// TIA Portal V16 export
// export: Created 2024-12-03T15:41:41.4210961Z, ExportSetting WithDefaults, DisplayName Totally Integrated Automation Portal, DisplayVersion V16 Update 6, DisplayName TIA Portal Version Control Interface, DisplayVersion V16 Update 2, DisplayName TIA Portal Openness, DisplayVersion V16 Update 6, DisplayName TIA Portal Teamcenter Gateway, DisplayVersion V16, DisplayName SINAMICS Startdrive Advanced, DisplayVersion V16 Update 5, DisplayName SINAMICS Startdrive G130, G150, S120, S150, SINAMICS MV, S210, DisplayVersion V16 Update 5, DisplayName SINAMICS Startdrive G110M, G120, G120C, G120D, G120P, G115D, DisplayVersion V16 Update 5, DisplayName STEP 7 Professional, DisplayVersion V16 Update 6, DisplayName STEP 7 Safety, DisplayVersion V16, DisplayName WinCC Advanced / Unified PC, DisplayVersion V16 Update 6
FUNCTION_BLOCK "CM_Encoder_FB"   // FB119, SCL
{ S7_Optimized_Access := 'TRUE' }
VERSION : 0.1
// stored: AutoNumber true, IsIECCheckEnabled false, IsRetainMemResEnabled false, MemoryReserve 100, SetENOAutomatically false, UDAEnableTagReadback false
   VAR_INPUT
      dEncr : DInt;   // Encoder input
      dPPR : DInt;   // Number of pulses per revolution
      rDiameterWheel : Real;   // Diameter of the wheel driving the roller or belt conveyor (mm)
      rGearRatio : Real;   // GearRatio should be 1.0 for the standalone encoders
      x32or16bitEncr : Bool;   // 1 = 32 bit, 0 = 16 bit
   END_VAR
   VAR_IN_OUT
      IO_Encoder : "VirtualEncoder_UDT";
   END_VAR
   VAR
      d16bitEncr_Range : DInt := 65535;   // Range of 16 bit encoder (pulses)
      d32bitEncr_Range : DInt;   // Range of 32 bit encoder (pulses)
      dCheckRotationClockwise : DInt;
      rPPmm : Real;   // # Pulses per mm
      rCircumference : Real;   // Contour of the driving wheel
      prevValue : DInt;
      currentValue : DInt;
      deltaPulses : DInt;
   END_VAR
BEGIN
   ////////////////////////////////////////////////////////////////////////////////////////////////////////////////
   //Processing encoder data
   ////////////////////////////////////////////////////////////////////////////////////////////////////////////////

   REGION Init
       #d16bitEncr_Range := 65535;
       #d32bitEncr_Range := 65536000 + 65535999;

   END_REGION

   REGION Update actual and old amount of pulses

       #prevValue := #currentValue;
       #currentValue := #dEncr;

   END_REGION

   REGION Calculate difference in amount of pulses (between 2 cycles)

       //Situation 1: From positive to negative sign
       IF #prevValue > 0 AND #currentValue < 0 THEN

           //Situation 1.1: Overflow detected 
           IF ABS(#currentValue - #prevValue) > (#d32bitEncr_Range / 2.0) AND #x32or16bitEncr THEN
               #deltaPulses := (#currentValue + #d32bitEncr_Range + 1) - #prevValue;
           ELSIF ABS(#currentValue - #prevValue) > (#d16bitEncr_Range / 2.0) AND NOT #x32or16bitEncr THEN
               #deltaPulses := (#currentValue + #d16bitEncr_Range + 1) - #prevValue;

               //Situation 1.2: No overflow (rotation not clockwise)    
           ELSE
               #deltaPulses := #currentValue - #prevValue;
           END_IF;

           //Situation 2: From negative to positive sign    
       ELSIF #prevValue < 0 AND #currentValue > 0 THEN

           //Situation 2.1: Overflow detected 
           IF ABS(#currentValue - #prevValue) > (#d32bitEncr_Range / 2.0) AND #x32or16bitEncr THEN
               #deltaPulses := (#currentValue - #d32bitEncr_Range - 1) - #prevValue;
           ELSIF ABS(#currentValue - #prevValue) > (#d16bitEncr_Range / 2.0) AND NOT #x32or16bitEncr THEN
               #deltaPulses := (#currentValue - #d16bitEncr_Range - 1) - #prevValue;

               //Situation 2.2: No overflow (rotation not clockwise)    
           ELSE
               #deltaPulses := #currentValue - #prevValue;
           END_IF;


           //Situation 3: no sign changes    
       ELSE
           #deltaPulses := #currentValue - #prevValue;

       END_IF;

   END_REGION

   REGION Convert # pulses to lineair distance (mm)
       #rPPmm := (#rDiameterWheel / 2.0) * ((2.0 * 3.14159265359) / DINT_TO_REAL(#dPPR));
       #IO_Encoder.Distance_mm := #rPPmm * #deltaPulses / #rGearRatio;

   END_REGION
END_FUNCTION_BLOCK
